FUNCTION_BLOCK PLOT_FROM_CSV
  {SET_ATTRIBUTE(OpcUa, SERVICE)}
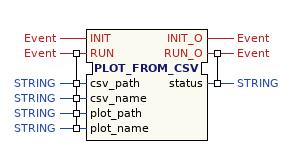
  EVENT_INPUT
    INIT;
    RUN WITH csv_path, csv_name, plot_path, plot_name; {SET_ATTRIBUTE(OpcUa, Method)}
  END_EVENT
  EVENT_OUTPUT
    INIT_O;
    RUN_O WITH status;
  END_EVENT
  VAR_INPUT
    csv_path : STRING; {SET_ATTRIBUTE(OpcUa, Variable.RUN)}
    csv_name : STRING; {SET_ATTRIBUTE(OpcUa, Variable.RUN)}
    plot_path : STRING; {SET_ATTRIBUTE(OpcUa, Variable.RUN)}
    plot_name : STRING; {SET_ATTRIBUTE(OpcUa, Variable.RUN)}
  END_VAR
  VAR_OUTPUT
    status : STRING; {SET_ATTRIBUTE(OpcUa, Variable.RUN)}
  END_VAR
END_FUNCTION_BLOCK
